TYPE MachineComRequest :
STRUCT
  Start : BOOL;
  Stop : BOOL;
  GoHome : BOOL;
  Halt : BOOL;
END_STRUCT
END_TYPE

(* stored: Version 1.1.0.1
   DUT MachineComRequest: Id {c8d6479a-0412-4bac-b9f3-3aefcc7bb8de} *)
